{attribute addProperty BoxType "APS4322-5000-0017"}
{attribute addProperty Id "FB_InputsAT %I*FB_Inputs_245CD1AC24643080WcStateAT %I*WcState_98A4DF7520.250InfoDataAT %I*InfoData_7231B2DD80100"}
{attribute addProperty CRC "2263788637"}
{attribute addProperty SizeInBites "2546"}
{attribute addProperty SizeInBytes "318.25"}
TYPE APS4322_59AFCAF5 :
STRUCT
	{attribute addProperty Name "FB_Inputs"}
	FB_Inputs : FB_Inputs_245CD1AC;
	{attribute addProperty Name "WcState"}
	WcState : WcState_98A4DF75;
	{attribute addProperty Name "InfoData"}
	InfoData : InfoData_7231B2DD;
END_STRUCT
END_TYPE

(* stored: Version 1.2.0.0, ProductVersion 3.1.4024.9
   DUT APS4322_59AFCAF5: Id {d0008498-1d9a-4b23-91e7-f6bceaea910a} *)
